{attribute addProperty BoxType "EK1122-0000-0018"}
{attribute addProperty Id "A_0060_AT2020_0250_0019_AT2020_0250A_0060_AT2020_0250_0019_AT2020_0250_DEA07AF962678.25Beckhoff_AT2xxxsub_EK1100EK1100_179A0949162A_0001_AT2000_0233_0022AT2000_1540501062678.25A_0002_AT2000_0233_0023AT2000_1540501062678.25A_0003_AT2000_0233_0024AT2000_1540501062678.25A_0004_AT2000_0250_0016AT2000_BA5A954865882.25A_0005_AT2000_0250_0017AT2000_BA5A954865882.25A_0006_AT2000_0250_0018AT2000_BA5A954865882.25A_0007_AT2000_0250_0019AT2000_BA5A954865882.25A_0008_AT2000_0250_0020AT2000_BA5A954865882.25A_0009_AT2000_0250_0021AT2000_BA5A954865882.25A_0010_AT2000_0250_0022AT2000_BA5A954865882.25A_0011_AT2000_0250_0023AT2000_BA5A954865882.25A_0012_AT2001_0250_0016AT2001_BA5A954865882.25A_0013_AT2001_0250_0017AT2001_BA5A954865882.25A_0014_AT2001_0250_0018AT2001_BA5A954865882.25A_0015_AT2001_0250_0019AT2001_BA5A954865882.25A_0016_AT2001_0250_0020AT2001_BA5A954865882.25A_0017_AT2001_0250_0022AT2001_BA5A954865882.25A_0018_AT2001_0250_0023AT2001_BA5A954865882.25A_0019_AT2001_0250_0024AT2001_BA5A954865882.25A_0020_AT2002_0249_0021AT2002_BA5A954865882.25A_0021_AT2002_0249_0022AT2002_BA5A954865882.25A_0022_AT2002_0249_0023AT2002_BA5A954865882.25A_0023_AT2002_0250_0022AT2002_BA5A954865882.25A_0024_AT2002_0250_0023AT2002_BA5A954865882.25A_0025_AT2002_0250_0024AT2002_BA5A954865882.25A_0026_AT2020_0250_0018AT2020_BA5A954865882.25A_0027_AT2020_0250_0021AT2020_BA5A954865882.25A_0028_AT2021_0250_0018AT2021_BA5A954865882.25A_0029_AT2021_0250_0020AT2021_BA5A954865882.25A_0030_AT2025_0250_0018AT2025_BA5A954865882.25A_0031_AT2026_0250_0021AT2026_BA5A954865882.25A_0032_AT2026_0250_0023AT2026_BA5A954865882.25A_0033_AT2040_0250_0018AT2040_BA5A954865882.25A_0034_AT2040_0250_0019AT2040_BA5A954865882.25A_0035_AT2040_0250_0020AT2040_BA5A954865882.25A_0036_AT2040_0250_0021A_0036_AT2040_0250_0021_A3885EBC62678.25A_0037_AT2040_0250_0022A_0037_AT2040_0250_0022_971D272D62678.25A_0038_AT2040_0250_0023A_0038_AT2040_0250_0023_2AEAC7B262678.25A_0039_AT2040_0250_0024A_0039_AT2040_0250_0024_A0FBBBF962678.25A_0040_AT2041_0250_0018A_0040_AT2041_0250_0018_599416E062678.25A_0041_AT2041_0250_0019A_0041_AT2041_0250_0019_45B99D7062678.25A_0042_AT2041_0250_0020A_0042_AT2041_0250_0020_B304CC6262678.25A_0043_AT2041_0250_0021A_0043_AT2041_0250_0021_3915B02962678.25A_0044_AT2041_0250_0022A_0044_AT2041_0250_0022_EA8B7A1C62678.25A_0045_AT2041_0250_0023A_0045_AT2041_0250_0023_5C753B7362678.25A_0046_AT2042_0250_0024A_0046_AT2042_0250_0024_35EBD52262678.25A_0047_AT2050_0500_0016A_0047_AT2050_0500_0016_017EACB362678.25A_0048_AT2050_0500_0017A_0048_AT2050_0500_0017_A8B58F1D62678.25A_0049_AT2050_0500_0018A_0049_AT2050_0500_0018_A5979C2D62678.25A_0050_AT2050_0500_0019A_0050_AT2050_0500_0019_E6F8155062678.25A_0051_AT2050_0500_0020A_0051_AT2050_0500_0020_6A24DD8862678.25A_0052_AT2050_0500_0021A_0052_AT2050_0500_0021_294B54F562678.25A_0053_AT2050_0500_0022A_0053_AT2050_0500_0022_49FE826D62678.25A_0054_AT2050_0500_0023A_0054_AT2050_0500_0023_9DD4EAFB62678.25A_0055_AT2050_0500_0024A_0055_AT2050_0500_0024_F6D8BACC62678.25A_0056_AT2050_0501_0017A_0056_AT2050_0501_0017_5F13996262678.25A_0057_AT2050_0501_0020A_0057_AT2050_0501_0020_6B86E0F362678.25A_0058_AT2050_0501_0021A_0058_AT2050_0501_0021_54B106B262678.25A_0061_AT2020_0250_0023_AT2020_0250A_0061_AT2020_0250_0023_AT2020_0250_0F2EDFD462678.25A_0062_AT2025_0250_0020_AT2025_0250A_0062_AT2025_0250_0020_AT2025_0250_1303544462678.25A_0063_AT2025_0250_0022_AT2025_0250A_0063_AT2025_0250_0022_AT2025_0250_9D18840C62678.25A_0064_AT2025_0250_0023_AT2025_0250A_0064_AT2025_0250_0023_AT2025_0250_4A8CE23A62678.25A_0065_AT2026_0250_0019_AT2026_0250A_0065_AT2026_0250_0019_AT2026_0250_E347C19462678.25A_0066_AT2026_0250_0020_AT2026_0250A_0066_AT2026_0250_0020_AT2026_0250_D7D2B80562678.25A_0067_AT2026_0250_0022_AT2026_0250A_0067_AT2026_0250_0022_AT2026_0250_D02FEC7062678.25A_0068_AT2026_0250_0024_AT2026_0250A_0068_AT2026_0250_0024_AT2026_0250_BF201DA562678.25A_0069_AT2050_0501_0019_AT2050_0501A_0069_AT2050_0501_0019_AT2050_0501_0D0F91BF62678.25A_0070_AT2050_0501_0022_AT2050_0501A_0070_AT2050_0501_0022_AT2050_0501_871EEDF462678.25A_0071_AT2050_0501_0023_AT2050_0501A_0071_AT2050_0501_0023_AT2050_0501_6B46D2C762678.25A_0072_AT2050_0501_0024_AT2050_0501A_0072_AT2050_0501_0024_AT2050_0501_776B595762678.25"}
{attribute addProperty CRC "1455759416"}
{attribute addProperty SizeInBites "45486"}
{attribute addProperty SizeInBytes "5685.75"}
TYPE Beckhoff_AT2xxxEK1122_56C52038 EXTENDS EK1122_179A0949 :
STRUCT
	{attribute addProperty Name "A_0060_AT2020_0250_0019_AT2020_0250"}
	A_0060_AT2020_0250_0019_AT2020_0250 : A_0060_AT2020_0250_0019_AT2020_0250_DEA07AF9;
	{attribute addProperty Name "Beckhoff_AT2xxxsub_EK1100"}
	Beckhoff_AT2xxxsub_EK1100 : EK1100_179A0949;
	{attribute addProperty Name "A_0001_AT2000_0233_0022"}
	A_0001_AT2000_0233_0022 : AT2000_15405010;
	{attribute addProperty Name "A_0002_AT2000_0233_0023"}
	A_0002_AT2000_0233_0023 : AT2000_15405010;
	{attribute addProperty Name "A_0003_AT2000_0233_0024"}
	A_0003_AT2000_0233_0024 : AT2000_15405010;
	{attribute addProperty Name "A_0004_AT2000_0250_0016"}
	A_0004_AT2000_0250_0016 : AT2000_BA5A9548;
	{attribute addProperty Name "A_0005_AT2000_0250_0017"}
	A_0005_AT2000_0250_0017 : AT2000_BA5A9548;
	{attribute addProperty Name "A_0006_AT2000_0250_0018"}
	A_0006_AT2000_0250_0018 : AT2000_BA5A9548;
	{attribute addProperty Name "A_0007_AT2000_0250_0019"}
	A_0007_AT2000_0250_0019 : AT2000_BA5A9548;
	{attribute addProperty Name "A_0008_AT2000_0250_0020"}
	A_0008_AT2000_0250_0020 : AT2000_BA5A9548;
	{attribute addProperty Name "A_0009_AT2000_0250_0021"}
	A_0009_AT2000_0250_0021 : AT2000_BA5A9548;
	{attribute addProperty Name "A_0010_AT2000_0250_0022"}
	A_0010_AT2000_0250_0022 : AT2000_BA5A9548;
	{attribute addProperty Name "A_0011_AT2000_0250_0023"}
	A_0011_AT2000_0250_0023 : AT2000_BA5A9548;
	{attribute addProperty Name "A_0012_AT2001_0250_0016"}
	A_0012_AT2001_0250_0016 : AT2001_BA5A9548;
	{attribute addProperty Name "A_0013_AT2001_0250_0017"}
	A_0013_AT2001_0250_0017 : AT2001_BA5A9548;
	{attribute addProperty Name "A_0014_AT2001_0250_0018"}
	A_0014_AT2001_0250_0018 : AT2001_BA5A9548;
	{attribute addProperty Name "A_0015_AT2001_0250_0019"}
	A_0015_AT2001_0250_0019 : AT2001_BA5A9548;
	{attribute addProperty Name "A_0016_AT2001_0250_0020"}
	A_0016_AT2001_0250_0020 : AT2001_BA5A9548;
	{attribute addProperty Name "A_0017_AT2001_0250_0022"}
	A_0017_AT2001_0250_0022 : AT2001_BA5A9548;
	{attribute addProperty Name "A_0018_AT2001_0250_0023"}
	A_0018_AT2001_0250_0023 : AT2001_BA5A9548;
	{attribute addProperty Name "A_0019_AT2001_0250_0024"}
	A_0019_AT2001_0250_0024 : AT2001_BA5A9548;
	{attribute addProperty Name "A_0020_AT2002_0249_0021"}
	A_0020_AT2002_0249_0021 : AT2002_BA5A9548;
	{attribute addProperty Name "A_0021_AT2002_0249_0022"}
	A_0021_AT2002_0249_0022 : AT2002_BA5A9548;
	{attribute addProperty Name "A_0022_AT2002_0249_0023"}
	A_0022_AT2002_0249_0023 : AT2002_BA5A9548;
	{attribute addProperty Name "A_0023_AT2002_0250_0022"}
	A_0023_AT2002_0250_0022 : AT2002_BA5A9548;
	{attribute addProperty Name "A_0024_AT2002_0250_0023"}
	A_0024_AT2002_0250_0023 : AT2002_BA5A9548;
	{attribute addProperty Name "A_0025_AT2002_0250_0024"}
	A_0025_AT2002_0250_0024 : AT2002_BA5A9548;
	{attribute addProperty Name "A_0026_AT2020_0250_0018"}
	A_0026_AT2020_0250_0018 : AT2020_BA5A9548;
	{attribute addProperty Name "A_0027_AT2020_0250_0021"}
	A_0027_AT2020_0250_0021 : AT2020_BA5A9548;
	{attribute addProperty Name "A_0028_AT2021_0250_0018"}
	A_0028_AT2021_0250_0018 : AT2021_BA5A9548;
	{attribute addProperty Name "A_0029_AT2021_0250_0020"}
	A_0029_AT2021_0250_0020 : AT2021_BA5A9548;
	{attribute addProperty Name "A_0030_AT2025_0250_0018"}
	A_0030_AT2025_0250_0018 : AT2025_BA5A9548;
	{attribute addProperty Name "A_0031_AT2026_0250_0021"}
	A_0031_AT2026_0250_0021 : AT2026_BA5A9548;
	{attribute addProperty Name "A_0032_AT2026_0250_0023"}
	A_0032_AT2026_0250_0023 : AT2026_BA5A9548;
	{attribute addProperty Name "A_0033_AT2040_0250_0018"}
	A_0033_AT2040_0250_0018 : AT2040_BA5A9548;
	{attribute addProperty Name "A_0034_AT2040_0250_0019"}
	A_0034_AT2040_0250_0019 : AT2040_BA5A9548;
	{attribute addProperty Name "A_0035_AT2040_0250_0020"}
	A_0035_AT2040_0250_0020 : AT2040_BA5A9548;
	{attribute addProperty Name "A_0036_AT2040_0250_0021"}
	A_0036_AT2040_0250_0021 : A_0036_AT2040_0250_0021_A3885EBC;
	{attribute addProperty Name "A_0037_AT2040_0250_0022"}
	A_0037_AT2040_0250_0022 : A_0037_AT2040_0250_0022_971D272D;
	{attribute addProperty Name "A_0038_AT2040_0250_0023"}
	A_0038_AT2040_0250_0023 : A_0038_AT2040_0250_0023_2AEAC7B2;
	{attribute addProperty Name "A_0039_AT2040_0250_0024"}
	A_0039_AT2040_0250_0024 : A_0039_AT2040_0250_0024_A0FBBBF9;
	{attribute addProperty Name "A_0040_AT2041_0250_0018"}
	A_0040_AT2041_0250_0018 : A_0040_AT2041_0250_0018_599416E0;
	{attribute addProperty Name "A_0041_AT2041_0250_0019"}
	A_0041_AT2041_0250_0019 : A_0041_AT2041_0250_0019_45B99D70;
	{attribute addProperty Name "A_0042_AT2041_0250_0020"}
	A_0042_AT2041_0250_0020 : A_0042_AT2041_0250_0020_B304CC62;
	{attribute addProperty Name "A_0043_AT2041_0250_0021"}
	A_0043_AT2041_0250_0021 : A_0043_AT2041_0250_0021_3915B029;
	{attribute addProperty Name "A_0044_AT2041_0250_0022"}
	A_0044_AT2041_0250_0022 : A_0044_AT2041_0250_0022_EA8B7A1C;
	{attribute addProperty Name "A_0045_AT2041_0250_0023"}
	A_0045_AT2041_0250_0023 : A_0045_AT2041_0250_0023_5C753B73;
	{attribute addProperty Name "A_0046_AT2042_0250_0024"}
	A_0046_AT2042_0250_0024 : A_0046_AT2042_0250_0024_35EBD522;
	{attribute addProperty Name "A_0047_AT2050_0500_0016"}
	A_0047_AT2050_0500_0016 : A_0047_AT2050_0500_0016_017EACB3;
	{attribute addProperty Name "A_0048_AT2050_0500_0017"}
	A_0048_AT2050_0500_0017 : A_0048_AT2050_0500_0017_A8B58F1D;
	{attribute addProperty Name "A_0049_AT2050_0500_0018"}
	A_0049_AT2050_0500_0018 : A_0049_AT2050_0500_0018_A5979C2D;
	{attribute addProperty Name "A_0050_AT2050_0500_0019"}
	A_0050_AT2050_0500_0019 : A_0050_AT2050_0500_0019_E6F81550;
	{attribute addProperty Name "A_0051_AT2050_0500_0020"}
	A_0051_AT2050_0500_0020 : A_0051_AT2050_0500_0020_6A24DD88;
	{attribute addProperty Name "A_0052_AT2050_0500_0021"}
	A_0052_AT2050_0500_0021 : A_0052_AT2050_0500_0021_294B54F5;
	{attribute addProperty Name "A_0053_AT2050_0500_0022"}
	A_0053_AT2050_0500_0022 : A_0053_AT2050_0500_0022_49FE826D;
	{attribute addProperty Name "A_0054_AT2050_0500_0023"}
	A_0054_AT2050_0500_0023 : A_0054_AT2050_0500_0023_9DD4EAFB;
	{attribute addProperty Name "A_0055_AT2050_0500_0024"}
	A_0055_AT2050_0500_0024 : A_0055_AT2050_0500_0024_F6D8BACC;
	{attribute addProperty Name "A_0056_AT2050_0501_0017"}
	A_0056_AT2050_0501_0017 : A_0056_AT2050_0501_0017_5F139962;
	{attribute addProperty Name "A_0057_AT2050_0501_0020"}
	A_0057_AT2050_0501_0020 : A_0057_AT2050_0501_0020_6B86E0F3;
	{attribute addProperty Name "A_0058_AT2050_0501_0021"}
	A_0058_AT2050_0501_0021 : A_0058_AT2050_0501_0021_54B106B2;
	{attribute addProperty Name "A_0061_AT2020_0250_0023_AT2020_0250"}
	A_0061_AT2020_0250_0023_AT2020_0250 : A_0061_AT2020_0250_0023_AT2020_0250_0F2EDFD4;
	{attribute addProperty Name "A_0062_AT2025_0250_0020_AT2025_0250"}
	A_0062_AT2025_0250_0020_AT2025_0250 : A_0062_AT2025_0250_0020_AT2025_0250_13035444;
	{attribute addProperty Name "A_0063_AT2025_0250_0022_AT2025_0250"}
	A_0063_AT2025_0250_0022_AT2025_0250 : A_0063_AT2025_0250_0022_AT2025_0250_9D18840C;
	{attribute addProperty Name "A_0064_AT2025_0250_0023_AT2025_0250"}
	A_0064_AT2025_0250_0023_AT2025_0250 : A_0064_AT2025_0250_0023_AT2025_0250_4A8CE23A;
	{attribute addProperty Name "A_0065_AT2026_0250_0019_AT2026_0250"}
	A_0065_AT2026_0250_0019_AT2026_0250 : A_0065_AT2026_0250_0019_AT2026_0250_E347C194;
	{attribute addProperty Name "A_0066_AT2026_0250_0020_AT2026_0250"}
	A_0066_AT2026_0250_0020_AT2026_0250 : A_0066_AT2026_0250_0020_AT2026_0250_D7D2B805;
	{attribute addProperty Name "A_0067_AT2026_0250_0022_AT2026_0250"}
	A_0067_AT2026_0250_0022_AT2026_0250 : A_0067_AT2026_0250_0022_AT2026_0250_D02FEC70;
	{attribute addProperty Name "A_0068_AT2026_0250_0024_AT2026_0250"}
	A_0068_AT2026_0250_0024_AT2026_0250 : A_0068_AT2026_0250_0024_AT2026_0250_BF201DA5;
	{attribute addProperty Name "A_0069_AT2050_0501_0019_AT2050_0501"}
	A_0069_AT2050_0501_0019_AT2050_0501 : A_0069_AT2050_0501_0019_AT2050_0501_0D0F91BF;
	{attribute addProperty Name "A_0070_AT2050_0501_0022_AT2050_0501"}
	A_0070_AT2050_0501_0022_AT2050_0501 : A_0070_AT2050_0501_0022_AT2050_0501_871EEDF4;
	{attribute addProperty Name "A_0071_AT2050_0501_0023_AT2050_0501"}
	A_0071_AT2050_0501_0023_AT2050_0501 : A_0071_AT2050_0501_0023_AT2050_0501_6B46D2C7;
	{attribute addProperty Name "A_0072_AT2050_0501_0024_AT2050_0501"}
	A_0072_AT2050_0501_0024_AT2050_0501 : A_0072_AT2050_0501_0024_AT2050_0501_776B5957;
END_STRUCT
END_TYPE

(* stored: Version 1.2.0.0, ProductVersion 3.1.4024.9
   DUT Beckhoff_AT2xxxEK1122_56C52038: Id {f12b503d-585f-4383-882c-b620e711f34a} *)
